PROGRAM INTERNAL MAIN
VAR
END_VAR

END_PROGRAM

(* stored: Version 1.1.0.1, ProductVersion 3.1.4026.18
   POU MAIN: Id {014aecf0-fb86-48d0-ad21-38693442dc4c}, SpecialFunc None *)
